Staubli VAL3: txt_PkgInit.pgx

program txt_PkgInit()
  local bool l_config
  local joint l_jTemp1
begin
  resetMotion()
  call Txt_initData()


  n_sTxt=0
  call TxtReadRoom1()
  if nTxtTotal>1
    call TxtReadRoom2()
  endIf
  l_config=pointToJoint(tTool,jConfig,pfrmCad[0],jConfig)

  bTxtPrSv=true
  sScrPts="OK"
  call hmi_refreshmain()
end
